(* Logix 5000 project; controller Beer_Brewing vendor 1 type 14 code 65 rev 20.18; software revision 20.06 *)

TASK MainTask (continuous, watchdog 500 ms) : MainProgram

MODULES
   Controller : vendor 1 type 14 code 65 (CompactLogixL35Controller 0, rev 20.18)
      LocalENB : 1769-L35E Ethernet Port (CompactLogixL35Ethernet 1, rev 20.11)
      Local : CompactBus (CompactVirtualAdapter 3, rev 20.11)
END_MODULES

VAR_GLOBAL   (* controller tags *)
   Add_Yeast : BOOL;
   Barley_Counter : COUNTER := (PRE := 28, DN := 1);
   Barley_Timer : TIMER := (PRE := 1000);
   Barley_Weight : REAL := 1400.0;   // Barley is added at 50kg/sec
   Brewing_Heater : BOOL;   // ON = 1 OFF = 0
   Brewing_Timer : TIMER := (PRE := 30000, EN := 1, DN := 1);
   BrewingKettle_Valve : BOOL;   // Open = 1 Closed = 0
   BrewingKettle_Valve_Closed : BOOL := 1;
   BrewingToWhirlpool_Pump : BOOL;   // ON = 1 OFF = 0
   BrewingToWhirlpool_Pump_Off : BOOL := 1;
   BrewingToWhirlpoolPump_Counter : COUNTER := (PRE := 70);
   BrewingToWhirlpoolPump_Timer : TIMER := (PRE := 1000);
   BrewingToWhirlpoolPumped_Gallons : REAL := 990.0;
   ColdWaterToHeatXchanger_Pump : BOOL;   // ON = 1 OFF = 0
   ConveyedMaltWeight : REAL := 1400.0;   // Malt Conveyed at 10 kg/sec
   Hops : BOOL;
   Hops_Timer : TIMER := (PRE := 5000, EN := 1, DN := 1);
   HotWater_Counter : COUNTER := (PRE := 66, DN := 1);
   HotWater_Timer : TIMER := (PRE := 1000);
   HotWaterPump_Off : BOOL := 1;
   HotWaterToMash_Pump : BOOL;   // ON = 1 OFF = 0
   LauterToBrewing_Pump : BOOL;   // ON = 1 OFF = 0
   LauterToBrewing_Pump_Off : BOOL := 1;
   LauterToBrewingPump_Counter : COUNTER := (PRE := 66, DN := 1);
   LauterToBrewingPump_Timer : TIMER := (PRE := 1000);
   LauterToBrewingPumped_Gallons : REAL := 990.0;
   LauterTun_Motor : BOOL;   // ON = 1 OFF = 0
   LauterTun_Valve : BOOL;   // Open = 1 Closed = 0
   LauterTun_Valve_Closed : BOOL := 1;
   LauterTunProcess_Timer : TIMER := (PRE := 15000, EN := 1, DN := 1);   // Set at 30 seconds (normally would be hours/days)
   Malt_Conveyor : BOOL;   // ON = 1 OFF = 0
   Malt_Counter : COUNTER := (PRE := 70, DN := 1);
   Malt_Heater : BOOL;   // ON = 1 OFF = 0
   Malt_Motor : BOOL;   // ON = 1 OFF = 0
   MaltConveyorOff_Timer : TIMER := (PRE := 20000, EN := 1, DN := 1);
   MaltDischargeTimer : TIMER := (PRE := 1000);
   Malting_Timer : TIMER := (PRE := 10000, EN := 1, DN := 1);
   MaltTank_Valve : BOOL;   // Open = 1 Closed = 0
   MaltValve_Close : BOOL := 1;
   Mash_Valve : BOOL;   // Open = 1 Closed = 0
   Mash_Valve_Closed : BOOL := 1;
   MashMotor : BOOL;   // ON = 1 OFF = 0
   MashMotorOff_Timer : TIMER := (PRE := 15000, EN := 1, DN := 1);
   MashToLauter_Pump : BOOL;   // ON = 1 OFF = 0
   MashToLauter_Pump_Off : BOOL := 1;
   MashToLauterPump_Counter : COUNTER := (PRE := 66, DN := 1);
   MashToLauterPump_Timer : TIMER := (PRE := 1000);
   MashToLauterPumped_Gallons : REAL := 990.0;
   Mill_Valve : BOOL;   // Open = 1 Closed = 0
   Milling_Motor : BOOL;   // ON = 1 OFF = 0
   MillingMotorOff_Timer : TIMER := (PRE := 30000, EN := 1, DN := 1);
   MillingProcessDone_Timer : TIMER := (PRE := 10000, EN := 1, DN := 1);
   MillToMash_Pump : BOOL;   // ON = 1 OFF = 0
   MillValve_Closed : BOOL := 1;
   PFToSFTank_Pump : BOOL;   // Pump from Primary Fermentation Tank to Secondary Fermentation Tank
   PFToSFTank_Pump_Off : BOOL := 1;
   PFToSFTankPump_Counter : COUNTER := (PRE := 70);
   PFToSFTankPump_Timer : TIMER := (PRE := 1000);
   PFToSFTankPumped_Gallons : REAL := 990.0;
   Powder_Counter : COUNTER := (PRE := 70, DN := 1);
   Powder_Timer : TIMER := (PRE := 1000);
   PowderPumpOff_Timer : TIMER := (PRE := 10000, EN := 1, DN := 1);
   PrimaryFermentationTank_Valve : BOOL;
   PrimaryFermentationTank_Valve_Closed : BOOL := 1;
   PrimaryFermentationTimer : TIMER := (PRE := 10000, EN := 1, DN := 1);
   ProcessON : BOOL;
   PumpedHotWater : REAL := 990.0;   // Hot water pumped at 15 gallons/sec
   PumpedPowderWeight : REAL := 1400.0;   // Powder pumped at 10kg/sec
   PumpedSproutWeight : REAL := 1400.0;
   PumpOFF : TIMER := (PRE := 7000, EN := 1, DN := 1);
   SecondaryFermentationTank_Valve : BOOL := 1;
   SecondaryFermentationTimer : TIMER := (PRE := 15000, EN := 1, DN := 1);   // Normally 3 months
   SFToFilter_Pump : BOOL := 1;   // Pump From Secondary Fermentation Tank to Filter
   Sprout_Counter : COUNTER := (PRE := 40, DN := 1);
   Sprout_Pump : BOOL;   // ON = 1 OFF = 0
   SproutDischargeTimer : TIMER := (PRE := 1000);
   Sprouting_Time : TIMER := (PRE := 10000, EN := 1, DN := 1);   // Time taken for sprouting (normally days)
   SproutTank_Valve : BOOL;   // Open = 1 Closed = 0
   SproutValve_Close : BOOL := 1;
   StartPB : BOOL;
   StopPB : BOOL;
   Water_Counter : COUNTER := (PRE := 14, DN := 1);
   Water_Gallons : REAL;   // Water is pumped at 15 gallons/sec
   Water_Timer : TIMER := (PRE := 1000);
   Whirlpool_Motor : BOOL;   // ON = 1 OFF = 0
   Whirlpool_Valve : BOOL;   // Open = 1 Closed = 0
   Whirlpool_Valve_Closed : BOOL := 1;
   WhirlpoolTimer : TIMER := (PRE := 15000, EN := 1, DN := 1);
   WhirlpoolToHeatXchanger_Pump : BOOL;   // ON = 1 OFF = 0
   WhirlpoolToHeatXchanger_Pump_Off : BOOL := 1;
   WhirlpoolToHeatXchangerPump_Counter : COUNTER := (PRE := 99, DN := 1);
   WhirlpoolToHeatXchangerPump_Timer : TIMER := (PRE := 1000);
   WhirlpoolToHeatXchangerPumped_Gallons : REAL := 990.0;   // Brew pumped at 10 gallons/sec
   YeastAddTimer : TIMER := (PRE := 8000, EN := 1, DN := 1);
END_VAR

PROGRAM MainProgram   (* main routine _00_MainRoutine *)

ROUTINE _00_MainRoutine   (* ladder *)
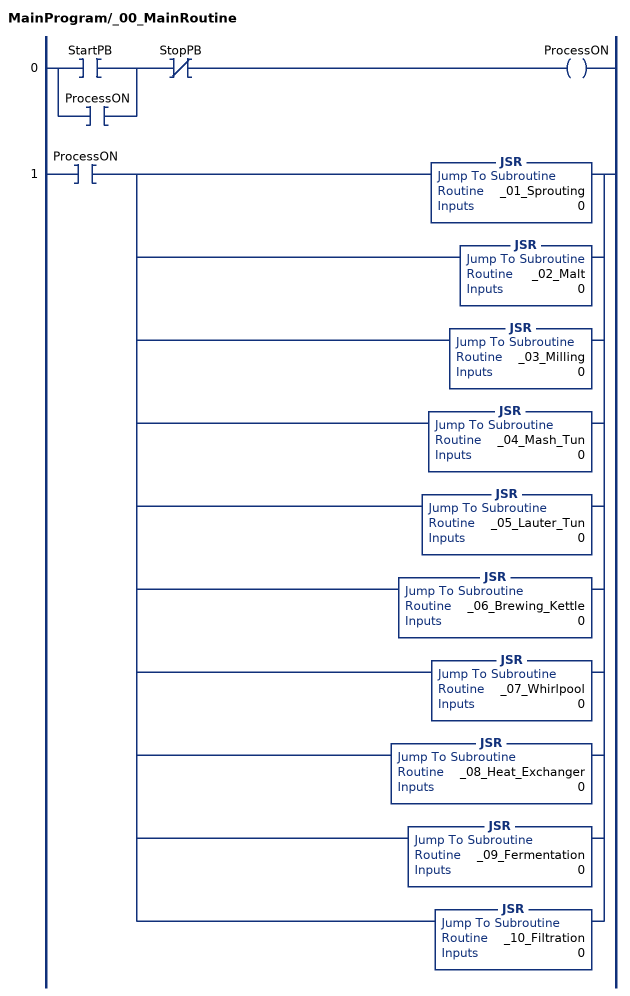
   0: [XIC(StartPB) ,XIC(ProcessON) ]XIO(StopPB)OTE(ProcessON);
   1: XIC(ProcessON)[JSR(_01_Sprouting,0) ,JSR(_02_Malt,0) ,JSR(_03_Milling,0) ,JSR(_04_Mash_Tun,0) ,JSR(_05_Lauter_Tun,0) ,JSR(_06_Brewing_Kettle,0) ,JSR(_07_Whirlpool,0) ,JSR(_08_Heat_Exchanger,0) ,JSR(_09_Fermentation,0) ,JSR(_10_Filtration,0) ];
END_ROUTINE

ROUTINE _01_Sprouting   (* ladder *)
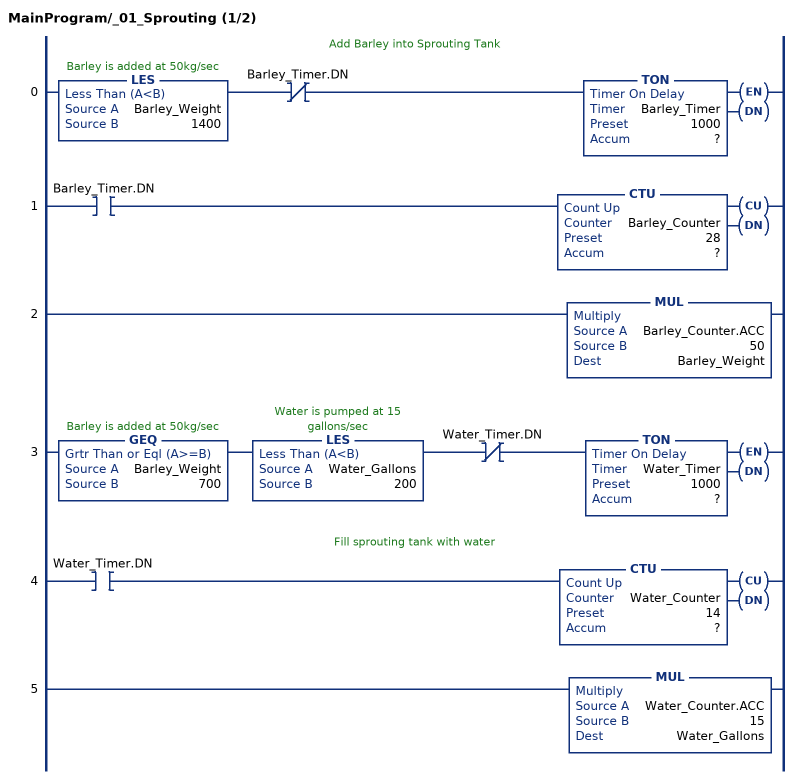
   // Add Barley into Sprouting Tank
   0: LES(Barley_Weight,1400)XIO(Barley_Timer.DN)TON(Barley_Timer,?,?);
   1: XIC(Barley_Timer.DN)CTU(Barley_Counter,?,?);
   2: MUL(Barley_Counter.ACC,50,Barley_Weight);
   3: GEQ(Barley_Weight,700)LES(Water_Gallons,200)XIO(Water_Timer.DN)TON(Water_Timer,?,?);
   // Fill sprouting tank with water
   4: XIC(Water_Timer.DN)CTU(Water_Counter,?,?);
   5: MUL(Water_Counter.ACC,15,Water_Gallons);
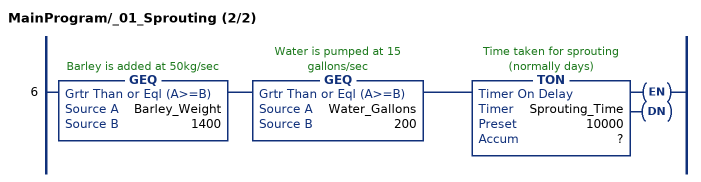
   6: GEQ(Barley_Weight,1400)GEQ(Water_Gallons,200)TON(Sprouting_Time,?,?);
END_ROUTINE

ROUTINE _02_Malt   (* ladder *)
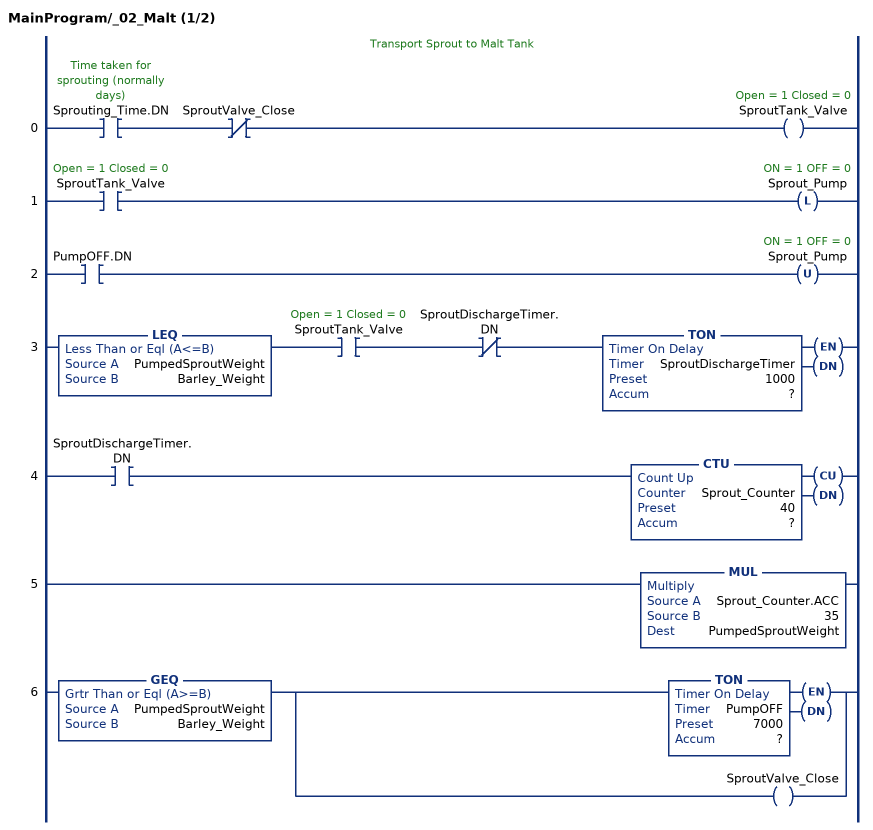
   // Transport Sprout to Malt Tank
   0: XIC(Sprouting_Time.DN)XIO(SproutValve_Close)OTE(SproutTank_Valve);
   1: XIC(SproutTank_Valve)OTL(Sprout_Pump);
   2: XIC(PumpOFF.DN)OTU(Sprout_Pump);
   3: LEQ(PumpedSproutWeight,Barley_Weight)XIC(SproutTank_Valve)XIO(SproutDischargeTimer.DN)TON(SproutDischargeTimer,?,?);
   4: XIC(SproutDischargeTimer.DN)CTU(Sprout_Counter,?,?);
   5: MUL(Sprout_Counter.ACC,35,PumpedSproutWeight);
   6: GEQ(PumpedSproutWeight,Barley_Weight)[TON(PumpOFF,?,?) ,OTE(SproutValve_Close) ];
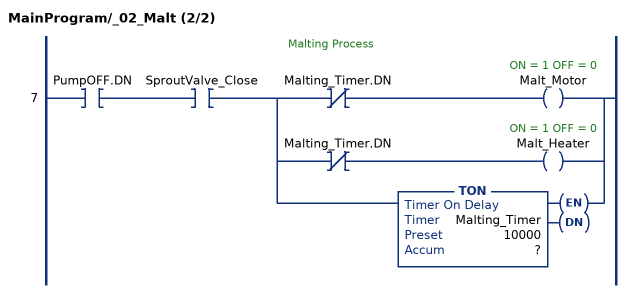
   // Malting Process
   7: XIC(PumpOFF.DN)XIC(SproutValve_Close)[XIO(Malting_Timer.DN) OTE(Malt_Motor) ,XIO(Malting_Timer.DN) OTE(Malt_Heater) ,TON(Malting_Timer,?,?) ];
END_ROUTINE

ROUTINE _03_Milling   (* ladder *)
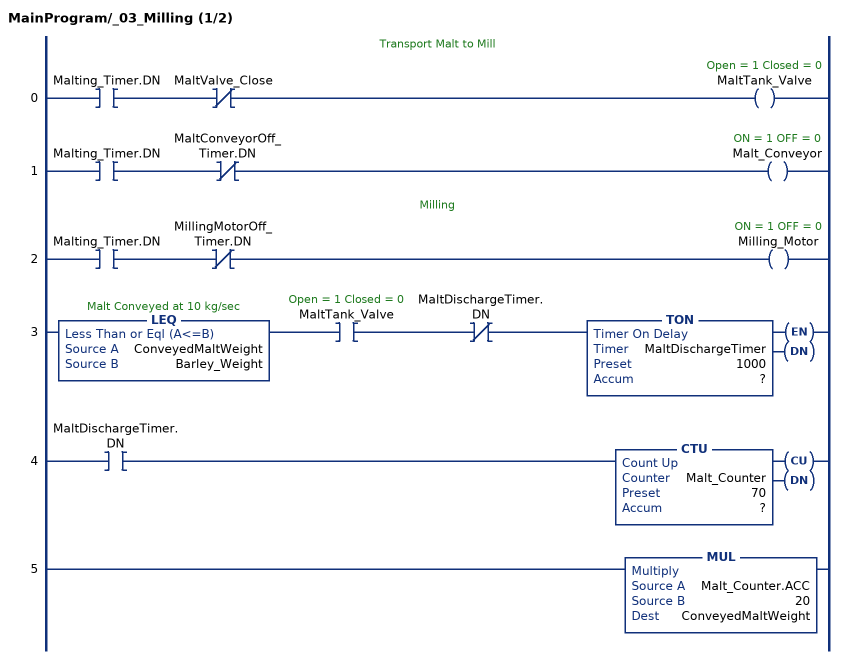
   // Transport Malt to Mill
   0: XIC(Malting_Timer.DN)XIO(MaltValve_Close)OTE(MaltTank_Valve);
   1: XIC(Malting_Timer.DN)XIO(MaltConveyorOff_Timer.DN)OTE(Malt_Conveyor);
   // Milling
   2: XIC(Malting_Timer.DN)XIO(MillingMotorOff_Timer.DN)OTE(Milling_Motor);
   3: LEQ(ConveyedMaltWeight,Barley_Weight)XIC(MaltTank_Valve)XIO(MaltDischargeTimer.DN)TON(MaltDischargeTimer,?,?);
   4: XIC(MaltDischargeTimer.DN)CTU(Malt_Counter,?,?);
   5: MUL(Malt_Counter.ACC,20,ConveyedMaltWeight);
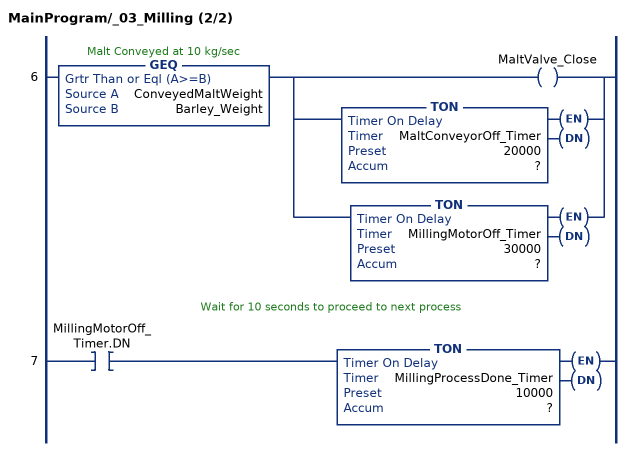
   6: GEQ(ConveyedMaltWeight,Barley_Weight)[OTE(MaltValve_Close) ,TON(MaltConveyorOff_Timer,?,?) ,TON(MillingMotorOff_Timer,?,?) ];
   // Wait for 10 seconds to proceed to next process
   7: XIC(MillingMotorOff_Timer.DN)TON(MillingProcessDone_Timer,?,?);
END_ROUTINE

ROUTINE _04_Mash_Tun   (* ladder *)
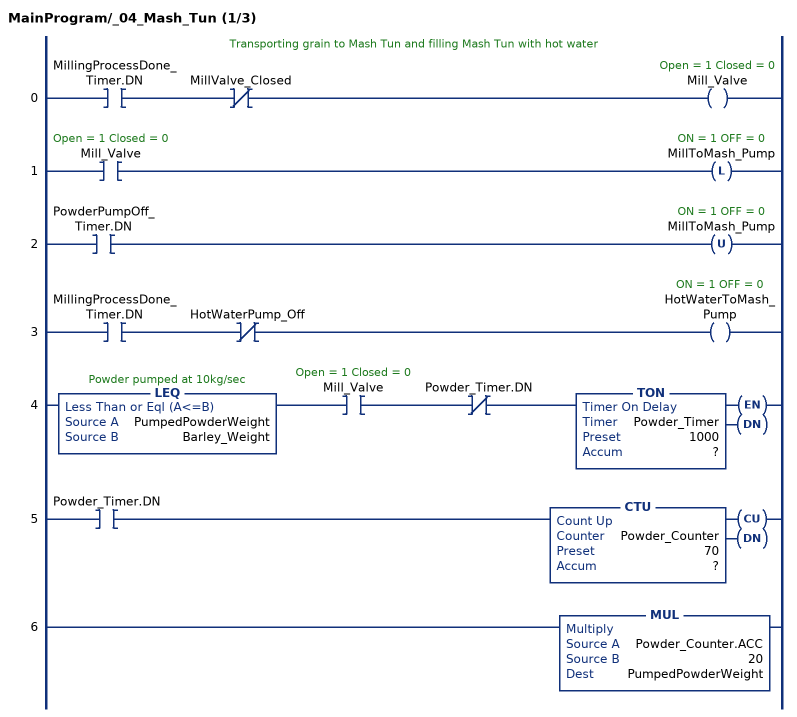
   // Transporting grain to Mash Tun and filling Mash Tun with hot water
   0: XIC(MillingProcessDone_Timer.DN)XIO(MillValve_Closed)OTE(Mill_Valve);
   1: XIC(Mill_Valve)OTL(MillToMash_Pump);
   2: XIC(PowderPumpOff_Timer.DN)OTU(MillToMash_Pump);
   3: XIC(MillingProcessDone_Timer.DN)XIO(HotWaterPump_Off)OTE(HotWaterToMash_Pump);
   4: LEQ(PumpedPowderWeight,Barley_Weight)XIC(Mill_Valve)XIO(Powder_Timer.DN)TON(Powder_Timer,?,?);
   5: XIC(Powder_Timer.DN)CTU(Powder_Counter,?,?);
   6: MUL(Powder_Counter.ACC,20,PumpedPowderWeight);
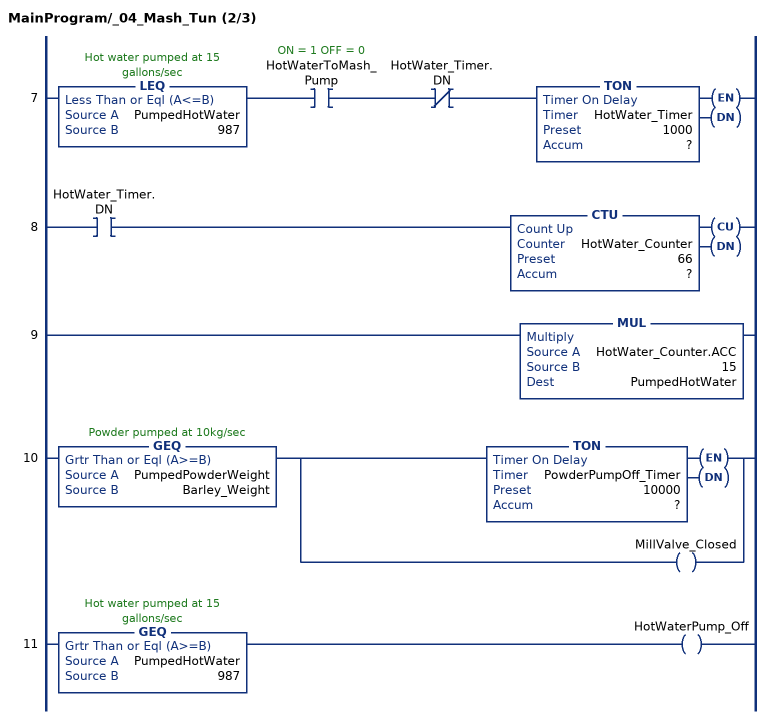
   7: LEQ(PumpedHotWater,987)XIC(HotWaterToMash_Pump)XIO(HotWater_Timer.DN)TON(HotWater_Timer,?,?);
   8: XIC(HotWater_Timer.DN)CTU(HotWater_Counter,?,?);
   9: MUL(HotWater_Counter.ACC,15,PumpedHotWater);
   10: GEQ(PumpedPowderWeight,Barley_Weight)[TON(PowderPumpOff_Timer,?,?) ,OTE(MillValve_Closed) ];
   11: GEQ(PumpedHotWater,987)OTE(HotWaterPump_Off);
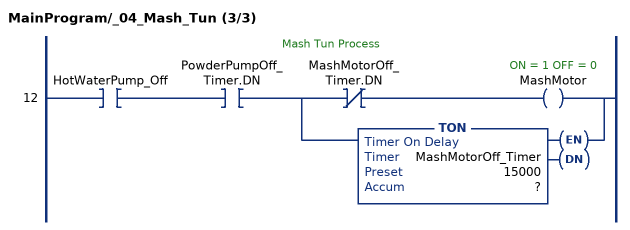
   // Mash Tun Process
   12: XIC(HotWaterPump_Off)XIC(PowderPumpOff_Timer.DN)[XIO(MashMotorOff_Timer.DN) OTE(MashMotor) ,TON(MashMotorOff_Timer,?,?) ];
END_ROUTINE

ROUTINE _05_Lauter_Tun   (* ladder *)
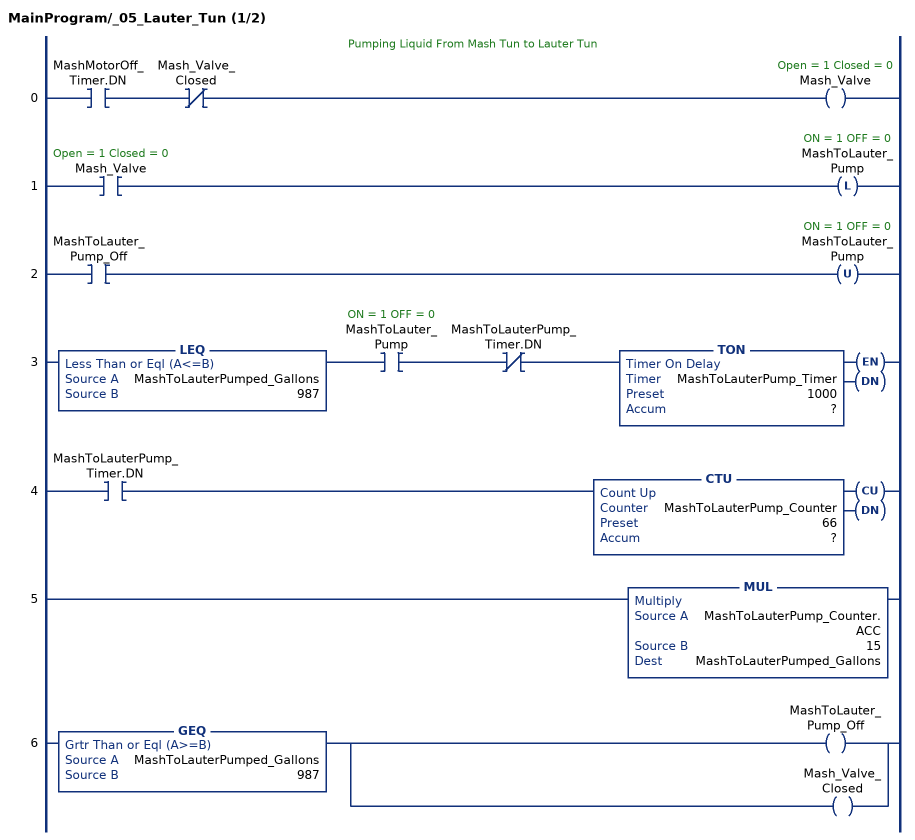
   // Pumping Liquid From Mash Tun to Lauter Tun
   0: XIC(MashMotorOff_Timer.DN)XIO(Mash_Valve_Closed)OTE(Mash_Valve);
   1: XIC(Mash_Valve)OTL(MashToLauter_Pump);
   2: XIC(MashToLauter_Pump_Off)OTU(MashToLauter_Pump);
   3: LEQ(MashToLauterPumped_Gallons,987)XIC(MashToLauter_Pump)XIO(MashToLauterPump_Timer.DN)TON(MashToLauterPump_Timer,?,?);
   4: XIC(MashToLauterPump_Timer.DN)CTU(MashToLauterPump_Counter,?,?);
   5: MUL(MashToLauterPump_Counter.ACC,15,MashToLauterPumped_Gallons);
   6: GEQ(MashToLauterPumped_Gallons,987)[OTE(MashToLauter_Pump_Off) ,OTE(Mash_Valve_Closed) ];
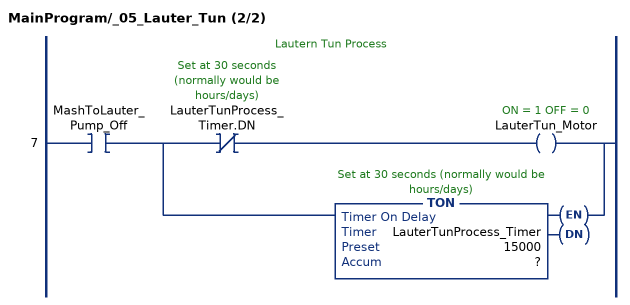
   // Lautern Tun Process
   7: XIC(MashToLauter_Pump_Off)[XIO(LauterTunProcess_Timer.DN) OTE(LauterTun_Motor) ,TON(LauterTunProcess_Timer,?,?) ];
END_ROUTINE

ROUTINE _06_Brewing_Kettle   (* ladder *)
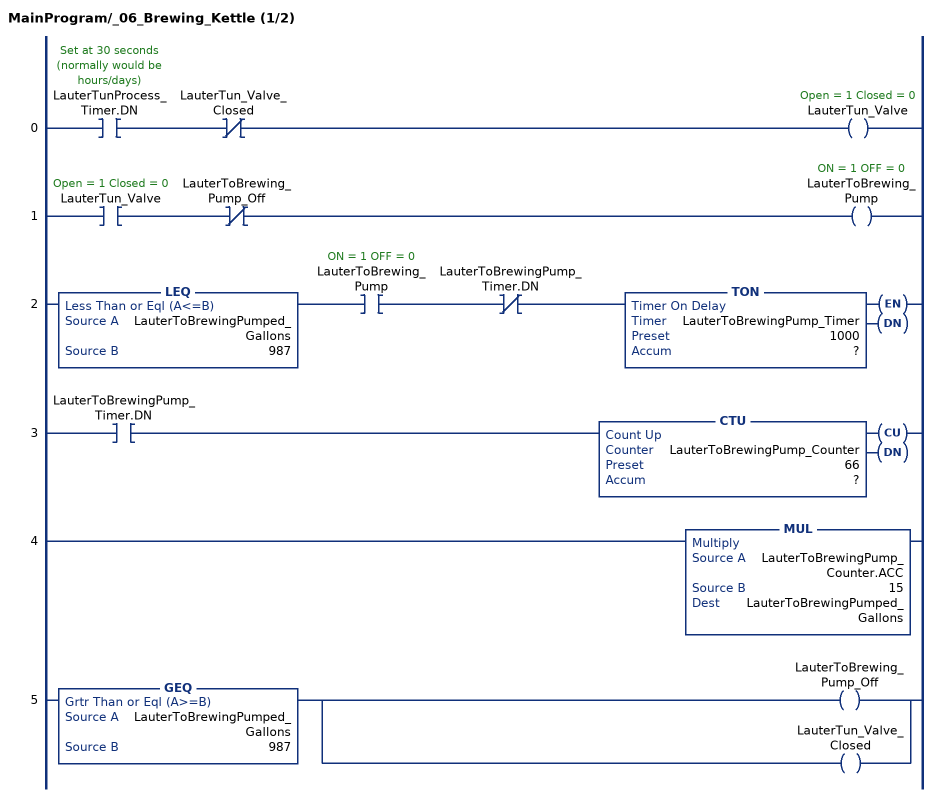
   0: XIC(LauterTunProcess_Timer.DN)XIO(LauterTun_Valve_Closed)OTE(LauterTun_Valve);
   1: XIC(LauterTun_Valve)XIO(LauterToBrewing_Pump_Off)OTE(LauterToBrewing_Pump);
   2: LEQ(LauterToBrewingPumped_Gallons,987)XIC(LauterToBrewing_Pump)XIO(LauterToBrewingPump_Timer.DN)TON(LauterToBrewingPump_Timer,?,?);
   3: XIC(LauterToBrewingPump_Timer.DN)CTU(LauterToBrewingPump_Counter,?,?);
   4: MUL(LauterToBrewingPump_Counter.ACC,15,LauterToBrewingPumped_Gallons);
   5: GEQ(LauterToBrewingPumped_Gallons,987)[OTE(LauterToBrewing_Pump_Off) ,OTE(LauterTun_Valve_Closed) ];
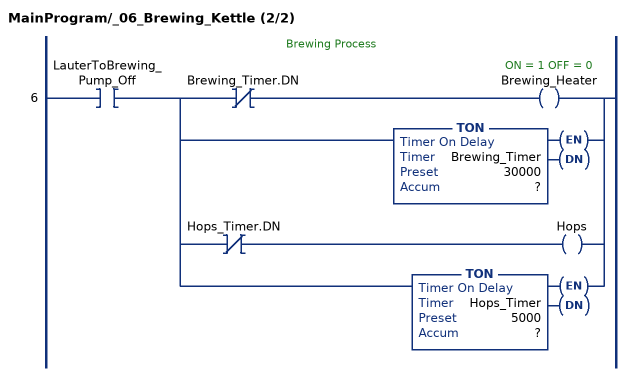
   // Brewing Process
   6: XIC(LauterToBrewing_Pump_Off)[XIO(Brewing_Timer.DN) OTE(Brewing_Heater) ,TON(Brewing_Timer,?,?) ,XIO(Hops_Timer.DN) OTE(Hops) ,TON(Hops_Timer,?,?) ];
END_ROUTINE

ROUTINE _07_Whirlpool   (* ladder *)
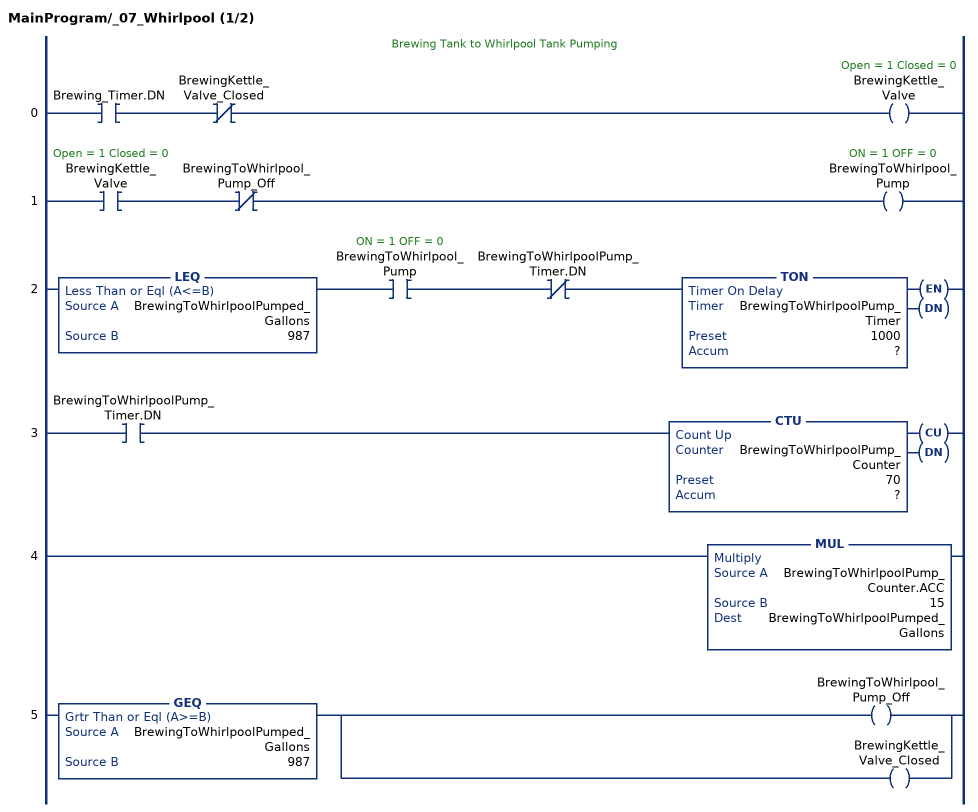
   // Brewing Tank to Whirlpool Tank Pumping
   0: XIC(Brewing_Timer.DN)XIO(BrewingKettle_Valve_Closed)OTE(BrewingKettle_Valve);
   1: XIC(BrewingKettle_Valve)XIO(BrewingToWhirlpool_Pump_Off)OTE(BrewingToWhirlpool_Pump);
   2: LEQ(BrewingToWhirlpoolPumped_Gallons,987)XIC(BrewingToWhirlpool_Pump)XIO(BrewingToWhirlpoolPump_Timer.DN)TON(BrewingToWhirlpoolPump_Timer,?,?);
   3: XIC(BrewingToWhirlpoolPump_Timer.DN)CTU(BrewingToWhirlpoolPump_Counter,?,?);
   4: MUL(BrewingToWhirlpoolPump_Counter.ACC,15,BrewingToWhirlpoolPumped_Gallons);
   5: GEQ(BrewingToWhirlpoolPumped_Gallons,987)[OTE(BrewingToWhirlpool_Pump_Off) ,OTE(BrewingKettle_Valve_Closed) ];
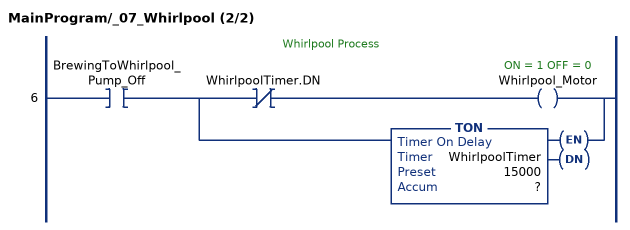
   // Whirlpool Process
   6: XIC(BrewingToWhirlpool_Pump_Off)[XIO(WhirlpoolTimer.DN) OTE(Whirlpool_Motor) ,TON(WhirlpoolTimer,?,?) ];
END_ROUTINE

ROUTINE _08_Heat_Exchanger   (* ladder *)
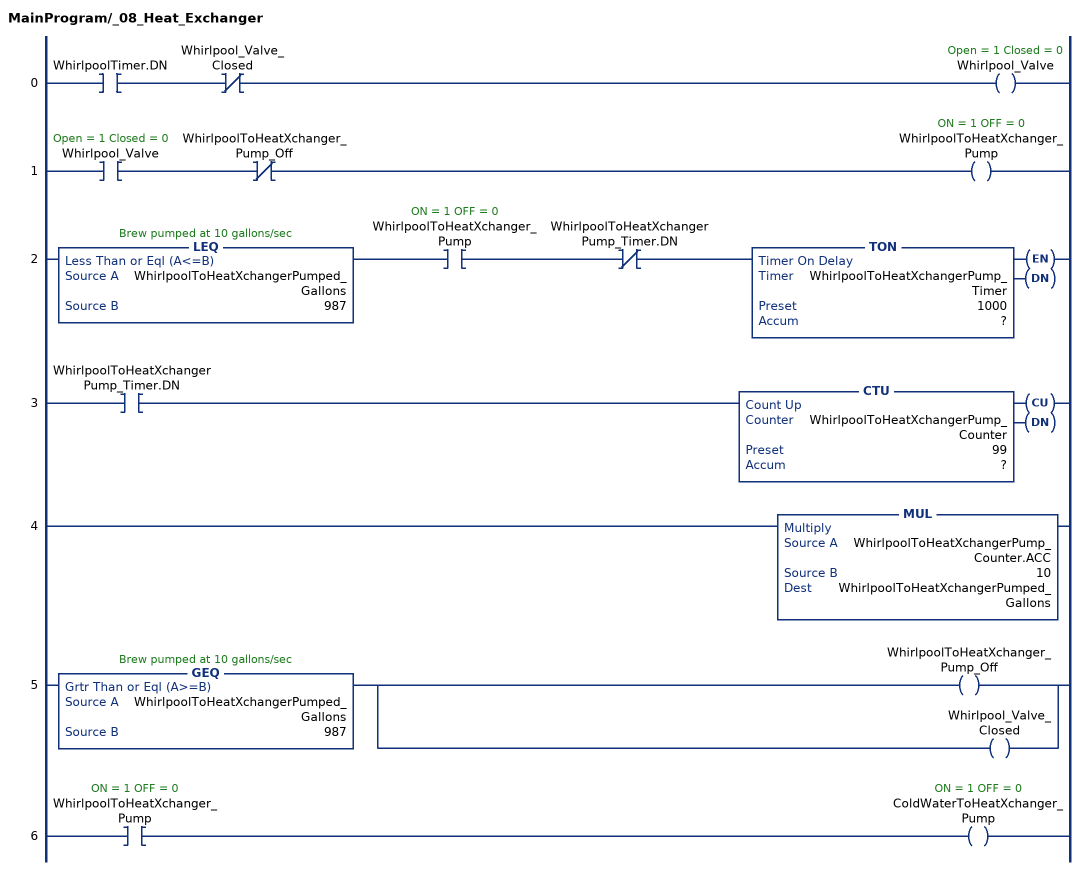
   0: XIC(WhirlpoolTimer.DN)XIO(Whirlpool_Valve_Closed)OTE(Whirlpool_Valve);
   1: XIC(Whirlpool_Valve)XIO(WhirlpoolToHeatXchanger_Pump_Off)OTE(WhirlpoolToHeatXchanger_Pump);
   2: LEQ(WhirlpoolToHeatXchangerPumped_Gallons,987)XIC(WhirlpoolToHeatXchanger_Pump)XIO(WhirlpoolToHeatXchangerPump_Timer.DN)TON(WhirlpoolToHeatXchangerPump_Timer,?,?);
   3: XIC(WhirlpoolToHeatXchangerPump_Timer.DN)CTU(WhirlpoolToHeatXchangerPump_Counter,?,?);
   4: MUL(WhirlpoolToHeatXchangerPump_Counter.ACC,10,WhirlpoolToHeatXchangerPumped_Gallons);
   5: GEQ(WhirlpoolToHeatXchangerPumped_Gallons,987)[OTE(WhirlpoolToHeatXchanger_Pump_Off) ,OTE(Whirlpool_Valve_Closed) ];
   6: XIC(WhirlpoolToHeatXchanger_Pump)OTE(ColdWaterToHeatXchanger_Pump);
END_ROUTINE

ROUTINE _09_Fermentation   (* ladder *)
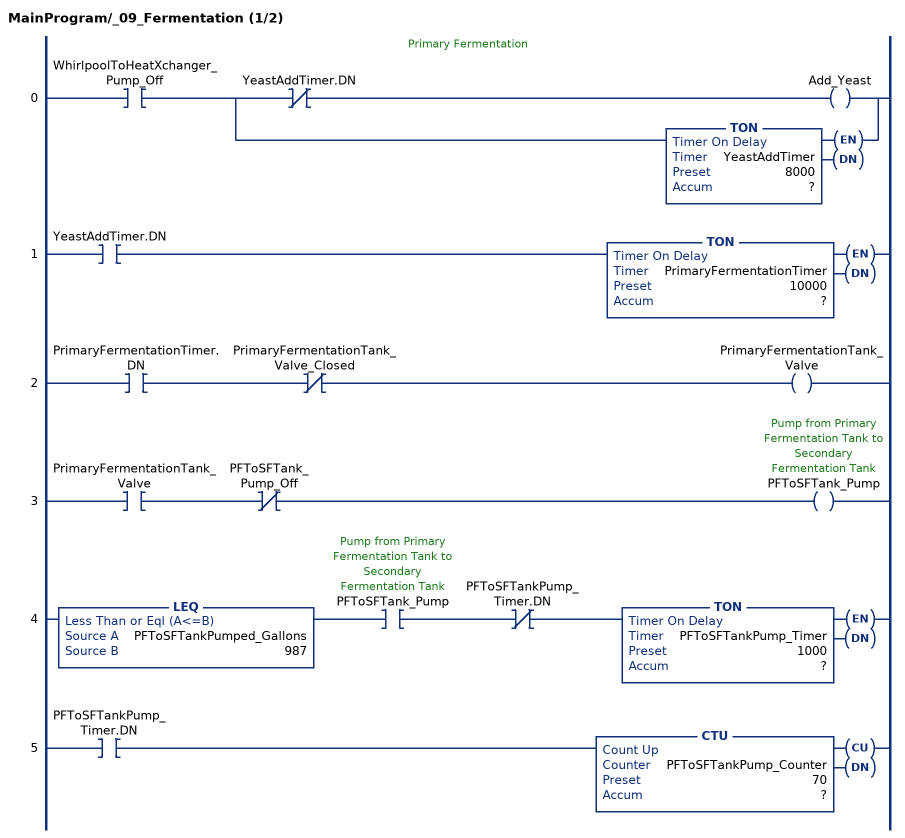
   // Primary Fermentation
   0: XIC(WhirlpoolToHeatXchanger_Pump_Off)[XIO(YeastAddTimer.DN) OTE(Add_Yeast) ,TON(YeastAddTimer,?,?) ];
   1: XIC(YeastAddTimer.DN)TON(PrimaryFermentationTimer,?,?);
   2: XIC(PrimaryFermentationTimer.DN)XIO(PrimaryFermentationTank_Valve_Closed)OTE(PrimaryFermentationTank_Valve);
   3: XIC(PrimaryFermentationTank_Valve)XIO(PFToSFTank_Pump_Off)OTE(PFToSFTank_Pump);
   4: LEQ(PFToSFTankPumped_Gallons,987)XIC(PFToSFTank_Pump)XIO(PFToSFTankPump_Timer.DN)TON(PFToSFTankPump_Timer,?,?);
   5: XIC(PFToSFTankPump_Timer.DN)CTU(PFToSFTankPump_Counter,?,?);
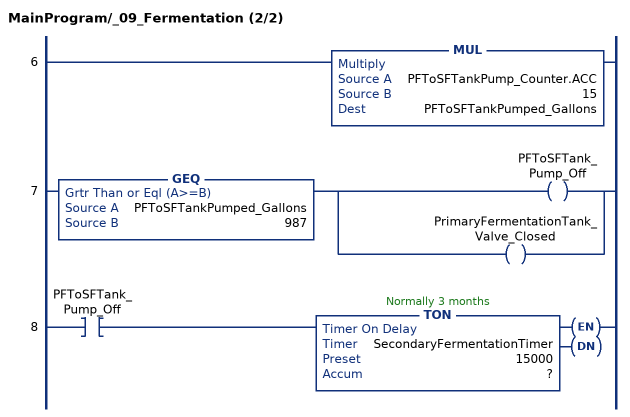
   6: MUL(PFToSFTankPump_Counter.ACC,15,PFToSFTankPumped_Gallons);
   7: GEQ(PFToSFTankPumped_Gallons,987)[OTE(PFToSFTank_Pump_Off) ,OTE(PrimaryFermentationTank_Valve_Closed) ];
   8: XIC(PFToSFTank_Pump_Off)TON(SecondaryFermentationTimer,?,?);
END_ROUTINE

ROUTINE _10_Filtration   (* ladder *)
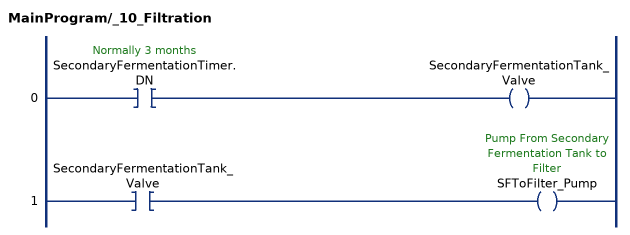
   0: XIC(SecondaryFermentationTimer.DN)OTE(SecondaryFermentationTank_Valve);
   1: XIC(SecondaryFermentationTank_Valve)OTE(SFToFilter_Pump);
END_ROUTINE
END_PROGRAM
